// TwinCAT 3 PLC project PLC
// Title: Test PLC project for ads-client library
// Company: Jussi Isotalo
// Author: Jussi Isotalo
// Description: Copyright (c) 2022 Jussi Isotalo <j.isotalo91@gmail.com> Permission is hereby granted, free of charge, to any person obtaining a copy of this software and associated documentation files (the "Software"), to deal in the Software without restriction, including without limitation the rights to use, copy, modify, merge, publish, distribute, sublicense, and/or sell copies of the Software, and to permit persons to whom the Software is furnished to do so, subject to the following conditions: The above copyright notice and this permission notice shall be included in all copies or substantial portions of the Software. THE SOFTWARE IS PROVIDED "AS IS", WITHOUT WARRANTY OF ANY KIND, EXPRESS OR IMPLIED, INCLUDING BUT NOT LIMITED TO THE WARRANTIES OF MERCHANTABILITY, FITNESS FOR A PARTICULAR PURPOSE AND NONINFRINGEMENT. IN NO EVENT SHALL THE AUTHORS OR COPYRIGHT HOLDERS BE LIABLE FOR ANY CLAIM, DAMAGES OR OTHER LIABILITY, WHETHER IN AN ACTION OF CONTRACT, TORT OR OTHERWISE, ARISING FROM, OUT OF OR IN CONNECTION WITH THE SOFTWARE OR THE USE OR OTHER DEALINGS IN THE SOFTWARE
// ProgramVersion: 3.1.4023.0
// libraries:
//   Tc2_DataExchange, * (Beckhoff Automation GmbH)
//   Tc2_Standard, * (Beckhoff Automation GmbH)
//   Tc2_System, * (Beckhoff Automation GmbH)
//   Tc2_Utilities, * (Beckhoff Automation GmbH)
//   Tc3_Module, * (Beckhoff Automation GmbH)
// project tree:
//   AdsClientTests/Data types/ FB_Block.TcPOU, FB_EmptyBlock.TcPOU, FB_EmptyBlock_1.TcPOU, I_Interface.TcIO, ST_Bits.TcDUT, ST_ComplexTypes_PackMode1.TcDUT, ST_ComplexTypes_PackMode8.TcDUT, ST_EmptyStruct.TcDUT (not stored), ST_IssueSpecificTypes.TcDUT, ST_SpecialTypes.TcDUT, ST_StandardTypes_PackMode1.TcDUT (not stored), ST_StandardTypes_PackMode8.TcDUT, ST_ComplexArrayTypes.TcDUT, E_Enum.TcDUT (not stored), E_LintEnum.TcDUT (not stored), StandardTypesAlias.TcDUT (not stored), ST_StandardTypes.TcDUT, ST_StandardArrayTypes.TcDUT (not stored), ST_ComplexTypes.TcDUT (not stored), U_Union.TcDUT (not stored)
//   AdsClientTests/ GVL_AdsClientTests.TcGVL, PRG_AdsClientTests.TcPOU
//   AdsClientTests/Read/ GVL_Read.TcGVL (not stored)
//   AdsClientTests/RPC/ FB_Rpc.TcPOU, GVL_RPC.TcGVL
//   AdsClientTests/Subscription/ GVL_Subscription.TcGVL, PRG_Subscription.TcPOU
//   AdsClientTests/Symbols and datatypes/ GVL_SymbolsAndDataTypes.TcGVL (not stored), ST_TestDataType.TcDUT (not stored)
//   AdsClientTests/Write/ GVL_Write.TcGVL
//   AdsClientTests/_OLD/ ST_Issue94.TcDUT, ST_Issue94_Byte.TcDUT, ST_PackMode1.TcDUT, ST_PackMode8.TcDUT, ST_Struct.TcDUT (not stored), ST_Struct2.TcDUT
//   / PlcTask.TcTTO (not stored)
// real-time tasks:
//   TASK PlcTask: cycle T#10ms, priority 20, ADS port 350
//   TASK PlcTask_852: cycle T#10ms, priority 21, ADS port 351

// ---- AdsClientTests/Data types/ST_Bits.TcDUT
TYPE ST_Bits :
STRUCT
	Bit_0 : BIT := TRUE;
	Bit_1 : BIT := FALSE;
	Bit_2 : BIT := FALSE;
	Bit_3 : BIT := TRUE;
	Bit_4 : BIT := TRUE;
	Bit_5 : BIT := FALSE;
	Bit_6 : BIT := FALSE;
	Bit_7 : BIT := TRUE;
	
	Bit_8 : BIT := FALSE;
	Bit_9 : BIT := TRUE;
	Bit_10 : BIT := TRUE;
	Bit_11 : BIT := FALSE;
	Bit_12 : BIT := FALSE;
	Bit_13 : BIT := TRUE;
	Bit_14 : BIT := TRUE;
	Bit_15 : BIT := FALSE;
	
	REAL_ : REAL := 3.14;
	
	Bit_16 : BIT := TRUE;
	Bit_17 : BIT := TRUE;
	Bit_18 : BIT := FALSE;
	Bit_19 : BIT := TRUE;
	Bit_20 : BIT := TRUE;
	Bit_21 : BIT := FALSE;
	Bit_22 : BIT := FALSE;
	Bit_23 : BIT := TRUE;
	
	Bit_24 : BIT := TRUE;
	Bit_25 : BIT := FALSE;
	Bit_26 : BIT := TRUE;
	Bit_27 : BIT := TRUE;
	Bit_28 : BIT := FALSE;
	Bit_29 : BIT := TRUE;
	Bit_30 : BIT := TRUE;
	Bit_31 : BIT := FALSE;
	
	Bit_32 : BIT := true;
END_STRUCT
END_TYPE

// ---- AdsClientTests/Data types/ST_ComplexTypes_PackMode1.TcDUT
{attribute 'pack_mode' := '1'}
TYPE ST_ComplexTypes_PackMode1 :
STRUCT
	STRUCT_ 	: ST_StandardTypes;
	STRUCT_2 	: ST_StandardArrayTypes;
	ALIAS_ 		: StandardTypesAlias;
	ENUM_		: E_Enum := E_Enum.Running;
	ENUM_2		: E_Enum := E_Enum.Unknown;
	ENUM_3		: E_Enum := 5555; //Not a valid value
	ENUM_4		: E_LintEnum := E_LintEnum.Negative;
	ENUM_5		: (Implicit, Enum, Values, Go, Here) := Values;
	POINTER_	: POINTER TO ST_StandardTypes;
	REFERENCE_	: REFERENCE TO ST_StandardTypes;
	SUBRANGE_	: INT(-4095..4095) := 1234;
	UNION_		: U_Union := (STRING_ := 'A test string ääöö!!@@'); 
	UNION_2		: U_Union := (INT_ := 32767); 
	UNION_3		: U_Union := (REAL_ := 3.14);
	BLOCK_		: FB_Block;
	BLOCK_2		: TON := (PT := T#2S500MS);
	BLOCK_3		: TC2_System.FB_CreateDir := (sPathName := 'C:\Test');
	BLOCK_4		: Tc2_DataExchange.FB_ReadAdsSymByName := (sVarName := 'GVL_Test.Variable');
	INTERFACE_	: I_Interface := BLOCK_;
END_STRUCT
END_TYPE

// ---- AdsClientTests/Data types/ST_ComplexTypes_PackMode8.TcDUT
{attribute 'pack_mode' := '1'}
TYPE ST_ComplexTypes_PackMode8 :
STRUCT
	STRUCT_ 	: ST_StandardTypes;
	STRUCT_2 	: ST_StandardArrayTypes;
	ALIAS_ 		: StandardTypesAlias;
	ENUM_		: E_Enum := E_Enum.Running;
	ENUM_2		: E_Enum := E_Enum.Unknown;
	ENUM_3		: E_Enum := 5555; //Not a valid value
	ENUM_4		: E_LintEnum := E_LintEnum.Negative;
	ENUM_5		: (Implicit, Enum, Values, Go, Here) := Values;
	POINTER_	: POINTER TO ST_StandardTypes;
	REFERENCE_	: REFERENCE TO ST_StandardTypes;
	SUBRANGE_	: INT(-4095..4095) := 1234;
	UNION_		: U_Union := (STRING_ := 'A test string ääöö!!@@'); 
	UNION_2		: U_Union := (INT_ := 32767); 
	UNION_3		: U_Union := (REAL_ := 3.14);
	BLOCK_		: FB_Block;
	BLOCK_2		: TON := (PT := T#2S500MS);
	BLOCK_3		: TC2_System.FB_CreateDir := (sPathName := 'C:\Test');
	BLOCK_4		: Tc2_DataExchange.FB_ReadAdsSymByName := (sVarName := 'GVL_Test.Variable');
	INTERFACE_	: I_Interface := BLOCK_;
END_STRUCT
END_TYPE

// ---- AdsClientTests/Data types/ST_IssueSpecificTypes.TcDUT
TYPE ST_IssueSpecificTypes :
STRUCT
	Issue94	: ST_Issue94;
END_STRUCT
END_TYPE

// ---- AdsClientTests/Data types/ST_SpecialTypes.TcDUT
TYPE ST_SpecialTypes :
STRUCT
	NegativeIndexArray		: ARRAY[-100..100] OF LREAL := [1.11, 99(0.0), 5.55, 99(0.0), 9.99];
	MultiDimensionalArray	: ARRAY[1..3, 1..2] OF BYTE := [1, 2, 3, 4, 5, 6];
	ArrayOfArrays			: ARRAY[1..3] OF ARRAY[1..2] OF SINT := [[-1, -2], [-3, -4], [-5, -6]];
	
	PackMode1		: ST_StandardTypes_PackMode1;
	PackMode1_2		: ST_ComplexTypes_PackMode1;
	PackMode8		: ST_StandardTypes_PackMode8;
	PackMode8_2		: ST_ComplexTypes_PackMode8;
	
	EmptyBlock		: FB_EmptyBlock;
	EmptyStruct		: ST_EmptyStruct;
	EmptyArray 		: ARRAY[0..-1] OF BOOL; //How is this even possible..?
	
	Bits			: ST_Bits;
END_STRUCT
END_TYPE

// ---- AdsClientTests/Data types/ST_StandardTypes_PackMode8.TcDUT
{attribute 'pack_mode' := '8'}
TYPE ST_StandardTypes_PackMode8:
STRUCT
	BOOL_ 	: BOOL := TRUE;
	BOOL_2 	: BOOL := FALSE;
	BYTE_ 	: BYTE := 255;
	WORD_ 	: WORD := 65535;
	DWORD_ 	: DWORD := 4294967295;
	SINT_ 	: SINT := 127;
	SINT_2 	: SINT := -128;
	USINT_ 	: USINT := 255;
	INT_ 	: INT := 32767;
	INT_2 	: INT := -32768;
	UINT_ 	: UINT := 65535;
	DINT_ 	: DINT := 2147483647;
	DINT_2 	: DINT := -2147483648;
	UDINT_ 	: UDINT := 4294967295;
	REAL_ 	: REAL := 3.4E38;
	REAL_2 	: REAL := -3.4E38;
	REAL_3 	: REAL := 75483.545;
	REAL_4 	: REAL := -75483.545;
	STRING_	: STRING := 'A test string ääöö!!@@';
	STRING_2: STRING(255) := 'Lorem ipsum dolor sit amet, consectetur adipiscing elit. Pellentesque bibendum mauris vel metus rutrum, sed gravida justo dignissim. Aenean et nisi cursus, auctor mi vel, posuere enim. Suspendisse ultricies mauris in finibus tristique. Nullam turpis duis.';
	DATE_ 	: DATE := D#2106-02-06;
	DT_ 	: DT := DT#2106-02-06-06:28:15;
	DT_2 	: DATE_AND_TIME := DT#2106-02-06-06:28:15;
	TOD_ 	: TOD := TO_TOD(4294967295);
	TOD_2 	: TIME_OF_DAY := TO_TOD(4294967295);
	TIME_ 	: TIME := T#49D17H2M47S295MS;
	LWORD_	: LWORD := 18446744073709551615;
	LINT_	: LINT := 9223372036854775807;
	LINT_2	: LINT := -9223372036854775808;
	ULINT_	: ULINT := 18446744073709551615;
	LREAL_ 	: LREAL := 1.7E308;
	LREAL_2 : LREAL := -1.7E308;
	LREAL_3 : REAL := 75483.545;
	LREAL_4 : REAL := -75483.545;
	WSTRING_: WSTRING := "A test wstring ääöö!!@@ ẞẟΔش";
	WSTRING_2: WSTRING(255) := "Lorem ipsum dolor sit amet, consectetur adipiscing elit. Pellentesque bibendum mauris vel metus rutrum, sed gravida justo dignissim. Aenean et nisi cursus, auctor mi vel, posuere enim. Suspendisse ultricies mauris in finibus tristique. Nullam turpis duis.";
	//LDATE_	: LDATE := LD#2554-7-21;
	//LDT_	: LDT := LDT#2554-7-21-23:34:33.709551615;
	//LTOD_	: LTOD := LTOD#23:59:59.999999999;
	LTIME_ 	: LTIME := LTIME#213503D23H34M33S709MS551US615NS;
END_STRUCT
END_TYPE

// ---- AdsClientTests/Data types/ST_ComplexArrayTypes.TcDUT
TYPE ST_ComplexArrayTypes :
STRUCT
	STRUCT_ 	: ARRAY[0..2] OF ST_StandardTypes;
	STRUCT_2 	: ARRAY[0..2] OF ST_StandardArrayTypes;
	ALIAS_ 		: ARRAY[0..2] OF StandardTypesAlias;
	ENUM_		: ARRAY[0..2] OF E_Enum := [E_Enum.Running, E_Enum.Disabled, E_Enum.Stopping];
	ENUM_2		: ARRAY[0..2] OF E_Enum := [E_Enum.Unknown, E_Enum.Disabled, E_Enum.Starting];
	ENUM_3		: ARRAY[0..2] OF E_Enum := [5555, 0, E_Enum.Unknown];
	ENUM_4		: ARRAY[0..2] OF E_LintEnum := [E_LintEnum.Negative, E_LintEnum.Zero, E_LintEnum.Positive];
	ENUM_5		: ARRAY[0..2] OF (Implicit, Enum, Values, Go, Here) := [2, 0, 4];
	POINTER_	: ARRAY[0..2] OF POINTER TO ST_StandardTypes;
	//REFERENCE_	: ARRAY[0..2] OF REFERENCE TO ST_StandardTypes;
	SUBRANGE_	: ARRAY[0..2] OF INT(-4095..4095) := [1234, 0, -1234];
	UNION_		: ARRAY[0..2] OF U_Union := [
		(STRING_ := 'A test string ääöö!!@@'),
		(INT_ := 32767),
		(REAL_ := 3.14)
	]; 
	BLOCK_		: ARRAY[0..2] OF FB_Block := [
		(StrValue := 'First'),
		(),
		(StrValue := 'Third')
	];
	BLOCK_2		: ARRAY[0..2] OF TON := [(PT := T#2S500MS), (), (PT := T#123S)];
	BLOCK_3		: ARRAY[0..2] OF TC2_System.FB_CreateDir := [
		(sPathName := 'C:\Test'),
		(),
		(sPathName := 'C:\AnotherTest')
	];
	BLOCK_4		: ARRAY[0..2] OF Tc2_DataExchange.FB_ReadAdsSymByName := [
		(sVarName := 'GVL_Test.Variable'),
		(),
		(sVarName := 'GVL_Test.AnotherVariable')
	];
	INTERFACE_	: ARRAY[0..2] OF I_Interface := [BLOCK_[0], 0, BLOCK_[2]];
END_STRUCT
END_TYPE

// ---- AdsClientTests/Data types/ST_StandardTypes.TcDUT
TYPE ST_StandardTypes :
STRUCT
	BOOL_ 	: BOOL := TRUE;
	BOOL_2 	: BOOL := FALSE;
	BYTE_ 	: BYTE := 255;
	WORD_ 	: WORD := 65535;
	DWORD_ 	: DWORD := 4294967295;
	SINT_ 	: SINT := 127;
	SINT_2 	: SINT := -128;
	USINT_ 	: USINT := 255;
	INT_ 	: INT := 32767;
	INT_2 	: INT := -32768;
	UINT_ 	: UINT := 65535;
	DINT_ 	: DINT := 2147483647;
	DINT_2 	: DINT := -2147483648;
	UDINT_ 	: UDINT := 4294967295;
	REAL_ 	: REAL := 3.4E38;
	REAL_2 	: REAL := -3.4E38;
	REAL_3 	: REAL := 75483.545;
	REAL_4 	: REAL := -75483.545;
	STRING_	: STRING := 'A test string ääöö!!@@';
	STRING_2: STRING(255) := 'Lorem ipsum dolor sit amet, consectetur adipiscing elit. Pellentesque bibendum mauris vel metus rutrum, sed gravida justo dignissim. Aenean et nisi cursus, auctor mi vel, posuere enim. Suspendisse ultricies mauris in finibus tristique. Nullam turpis duis.';
	DATE_ 	: DATE := D#2106-02-06;
	DT_ 	: DT := DT#2106-02-06-06:28:15;
	DT_2 	: DATE_AND_TIME := DT#2106-02-06-06:28:15;
	TOD_ 	: TOD := TO_TOD(4294967295);
	TOD_2 	: TIME_OF_DAY := TO_TOD(4294967295);
	TIME_ 	: TIME := T#49D17H2M47S295MS;
	LWORD_	: LWORD := 18446744073709551615;
	LINT_	: LINT := 9223372036854775807;
	LINT_2	: LINT := -9223372036854775808;
	ULINT_	: ULINT := 18446744073709551615;
	LREAL_ 	: LREAL := 1.7E308;
	LREAL_2 : LREAL := -1.7E308;
	LREAL_3 : REAL := 75483.545;
	LREAL_4 : REAL := -75483.545;
	WSTRING_: WSTRING := "A test wstring ääöö!!@@ ẞẟΔش";
	WSTRING_2: WSTRING(255) := "Lorem ipsum dolor sit amet, consectetur adipiscing elit. Pellentesque bibendum mauris vel metus rutrum, sed gravida justo dignissim. Aenean et nisi cursus, auctor mi vel, posuere enim. Suspendisse ultricies mauris in finibus tristique. Nullam turpis duis.";
	//LDATE_	: LDATE := LD#2554-7-21;
	//LDT_	: LDT := LDT#2554-7-21-23:34:33.709551615;
	//LTOD_	: LTOD := LTOD#23:59:59.999999999;
	LTIME_ 	: LTIME := LTIME#213503D23H34M33S709MS551US615NS;
END_STRUCT
END_TYPE

// ---- AdsClientTests/_OLD/ST_Issue94.TcDUT
TYPE ST_Issue94 :
STRUCT
	BoolValue 	: bool := TRUE;
	ArrayValue 	:  ARRAY [0..1] OF ST_Issue94_Byte := [(ByteValue := 1), (ByteValue := 2)];
END_STRUCT
END_TYPE

// ---- AdsClientTests/_OLD/ST_Issue94_Byte.TcDUT
TYPE ST_Issue94_Byte :
STRUCT
	ByteValue : byte;
END_STRUCT
END_TYPE

// ---- AdsClientTests/_OLD/ST_PackMode1.TcDUT
{attribute 'pack_mode' := '1'}
TYPE ST_PackMode1 :
STRUCT
	BoolValue 	: BOOL := TRUE;
	StringValue : STRING(27) := 'A string value';
	LrealValue 	: LREAL := 12321.3123123;
	BoolArray 	: ARRAY[1..5] OF BOOL;
	BlockArray 	: ARRAY[1..5] OF r_trig;
	LargeBlock 	: Tc2_System.FB_FileOpen := (sPathName := 'test_path');
END_STRUCT
END_TYPE

// ---- AdsClientTests/_OLD/ST_PackMode8.TcDUT
{attribute 'pack_mode' := '8'}
TYPE ST_PackMode8 :
STRUCT
	BoolValue 	: BOOL := TRUE;
	StringValue : STRING(27) := 'A string value';
	LrealValue 	: LREAL := 12321.3123123;
	BoolArray 	: ARRAY[1..5] OF BOOL;
	BlockArray 	: ARRAY[1..5] OF r_trig;
	LargeBlock 	: Tc2_System.FB_FileOpen := (sPathName := 'test_path');
END_STRUCT
END_TYPE

// ---- AdsClientTests/_OLD/ST_Struct2.TcDUT
TYPE ST_Struct2 :
STRUCT
	BoolValue 	: BOOL := TRUE;
	StringValue : STRING(27) := 'A string value';
	LrealValue 	: LREAL := 12321.3123123;
	BoolArray 	: ARRAY[1..5] OF BOOL := [TRUE, FALSE, TRUE, FALSE, TRUE];
	SubStruct	: ST_Struct;
END_STRUCT
END_TYPE

// ---- AdsClientTests/GVL_AdsClientTests.TcGVL
{attribute 'qualified_only'}
VAR_GLOBAL
	VERSION			: STRING := '2.0.0';
	IsReset 		: BOOL := TRUE;
	IsTestProject 	: BOOL := TRUE;
	IsRunning 		: BOOL;
	TestPointer 	: POINTER TO BOOL; //For 32/64bit check
END_VAR

// ---- AdsClientTests/RPC/GVL_RPC.TcGVL
{attribute 'qualified_only'}
VAR_GLOBAL
	RpcBlock : FB_Rpc;
	
END_VAR

// ---- AdsClientTests/Subscription/GVL_Subscription.TcGVL
{attribute 'qualified_only'}
VAR_GLOBAL
	NumericValue_10ms : INT;
	NumericValue_100ms : INT;
	NumericValue_1000ms : INT;
	Numericvalue_Constant : INT := 12245;
	
	BoolValue			: BOOL;
	StringValue       	: STRING;
	StructValue     	: ST_Struct;
END_VAR

// ---- AdsClientTests/Write/GVL_Write.TcGVL
{attribute 'qualified_only'}
VAR_GLOBAL
	StandardTypes 		: ST_StandardTypes;
	StandardArrays 		: ST_StandardArrayTypes;
	ComplexTypes		: ST_ComplexTypes := (
		POINTER_ 	:= ADR(StandardTypes),
		REFERENCE_ 	:= StandardTypes 
	);
	ComplexArrayTypes	: ST_ComplexArrayTypes;
	SpecialTypes		: ST_SpecialTypes;
	IssueSpecificTypes	: ST_IssueSpecificTypes;
	
END_VAR

// ---- AdsClientTests/Data types/I_Interface.TcIO
INTERFACE I_Interface

END_INTERFACE

// ---- AdsClientTests/RPC/FB_Rpc.TcPOU
FUNCTION_BLOCK FB_Rpc
VAR_INPUT
END_VAR
VAR_OUTPUT
END_VAR
VAR
END_VAR

{attribute 'TcRpcEnable'}
METHOD Calculator : BOOL
VAR_INPUT
	Value1	: REAL;
	Value2	: REAL;
END_VAR
VAR_OUTPUT
	Sum			: REAL;
	Product 	: REAL;
	Division	: REAL;
END_VAR
//Return TRUE if all success
Calculator := TRUE;

Sum := Value1 + Value2;
Product := Value1 * Value2;

IF Value2 <> 0 THEN
	Division := Value1 / Value2;
ELSE
	Division := 0;
	Calculator := FALSE;
END_IF
END_METHOD

{attribute 'TcRpcEnable'}
METHOD StructTest : ST_Struct
VAR_INPUT
	Input	: ST_Struct;
END_VAR
StructTest.SomeText := CONCAT('Response: ', Input.SomeText);
StructTest.SomeReal := Input.SomeReal * 10.0;
StructTest.SomeDate := Input.SomeDate + T#24H;
END_METHOD

END_FUNCTION_BLOCK

// ---- AdsClientTests/Data types/FB_Block.TcPOU
FUNCTION_BLOCK FB_Block IMPLEMENTS I_Interface
VAR_INPUT
END_VAR
VAR_OUTPUT
END_VAR
VAR
	StrValue : string;
	Data : ST_StandardTypes;
END_VAR

END_FUNCTION_BLOCK

// ---- AdsClientTests/Data types/FB_EmptyBlock.TcPOU
FUNCTION_BLOCK FB_EmptyBlock
VAR_INPUT
END_VAR
VAR_OUTPUT
END_VAR
VAR
END_VAR

END_FUNCTION_BLOCK

// ---- AdsClientTests/Data types/FB_EmptyBlock_1.TcPOU
FUNCTION_BLOCK FB_EmptyBlock_1
VAR_INPUT
END_VAR
VAR_OUTPUT
END_VAR
VAR
	value : BOOL;
END_VAR

END_FUNCTION_BLOCK

// ---- AdsClientTests/PRG_AdsClientTests.TcPOU
PROGRAM PRG_AdsClientTests
VAR
	InitDone : bool;
END_VAR

IF NOT GVL_AdsClientTests.IsRunning THEN
	MEMSET(ADR(GVL_Write.StandardTypes), 0, SIZEOF(GVL_Write.StandardTypes));
	MEMSET(ADR(GVL_Write.StandardTypes), 0, SIZEOF(GVL_Write.StandardArrays));
	MEMSET(ADR(GVL_Write.ComplexTypes), 0, SIZEOF(GVL_Write.ComplexTypes));
	MEMSET(ADR(GVL_Write.ComplexArrayTypes), 0, SIZEOF(GVL_Write.ComplexArrayTypes));
	MEMSET(ADR(GVL_Write.SpecialTypes), 0, SIZEOF(GVL_Write.SpecialTypes));
	MEMSET(ADR(GVL_Write.IssueSpecificTypes), 0, SIZEOF(GVL_Write.IssueSpecificTypes));
	
	GVL_Write.ComplexTypes.POINTER_ := ADR(GVL_Write.StandardTypes);
	GVL_Write.ComplexTypes.REFERENCE_ ref= GVL_Write.StandardTypes;
	
	GVL_AdsClientTests.IsRunning := TRUE;
END_IF

PRG_Subscription();

END_PROGRAM

// ---- AdsClientTests/Subscription/PRG_Subscription.TcPOU
PROGRAM PRG_Subscription
VAR
END_VAR

END_PROGRAM
